PROGRAM MAIN
VAR
	linkedList_TestSuite : LinkedList_TestSuite;
	queue_TestSuite : Queue_TestSuite;
	stack_TestSuite : Stack_TestSuite;
	forwardEnumerator_TestSuite : ForwardEnumerator_TestSuite;
	collection_TestSuite : Collection_TestSuite;
	_list_TestSuite : List_TestSuite;
	_listEnumerator_TestSuite : ListEnumerator_TestSuite;
	
	// variables used in examples	teset
	linkedList : LinkedList;
	queue : Queue;
	stack : Stack;
	value1 : INT := 123;
	value2 : INT := 456;
	value3 : INT := 789;
	enumerator : I_ForwardEnumerator;
	output : INT;
	allowed : BOOL;
END_VAR

TcUnit.RUN();

// LinkedList Examples
// ===================

// using AddFirst, First and RemoveFirst
// -------------------------------------

linkedList.AddFirst(value1); // (first->) 123 (<-last)
linkedList.AddFirst(value2); // (first->) 456, 123 (<-last)
linkedList.AddFirst(value3); // (first->) 789, 456, 123  (<-last)

enumerator := linkedList.GetEnumerator();
// the enumerator follows the .net style, which means you must call MoveNext once to
// move to the first item.  This allows you to directly use the enumerator in a while
// loop.
WHILE enumerator.MoveNext() DO
	enumerator.TryGet(output); // 1st pass output = 789, 2nd pass output = 456, 3rd pass output = 123
END_WHILE;
// you must dispose enumerators as they are new objects.
enumerator.Dispose();

allowed := linkedList.First.TryGet(output); // allowed = true, output = 789
linkedList.RemoveFirst(); // (first->) 456, 123  (<-last)
allowed := linkedList.First.TryGet(output); // allowed = true, output = 456
linkedList.RemoveFirst(); // (first->) 123  (<-last)
allowed := linkedList.First.TryGet(output); // allowed = true, output = 123
linkedList.RemoveFirst(); // (first->) null (<-last)

// Queue Examples
// ==============

// using Enqueue, TryPeek and TryDequeue
// -------------------------------------

queue.Enqueue(value1); // (first->) 123
queue.Enqueue(value2); // (first->) 123, 456
queue.Enqueue(value3); // (first->) 123, 456, 789

// TryPeek will not remove the item from the queue
allowed := queue.TryPeek(output); // allowed = true, output = 123

// TryDequeue will remove the item from the queue
allowed := queue.TryDequeue(output); // allowed = true, output = 123
allowed := queue.TryDequeue(output); // allowed = true, output = 456
allowed := queue.TryDequeue(output); // allowed = true, output = 789

// Stack Examples
// ==============

// using Push, TryPeek and TryPop
// -------------------------------------

stack.Push(value1); // (fifo->) 123
stack.Push(value2); // (fifo->) 456, 123
stack.Push(value3); // (fifo->) 789, 456, 123

// TryPeek will not remove the item from the stack
allowed := stack.TryPeek(output); // allowed = true, output = 789

// TryDequeue will remove the item from the queue
allowed := stack.TryPop(output); // allowed = true, output = 789
allowed := stack.TryPop(output); // allowed = true, output = 456
allowed := stack.TryPop(output); // allowed = true, output = 123

END_PROGRAM

(* stored: Version 1.1.0.1, ProductVersion 3.1.4024.12
   POU MAIN: Id {4fc6a7e2-9479-48b5-85ef-622583cb9cd0}, SpecialFunc None *)
